DATA_BLOCK "DB_OrinCommandValidation"
{ S7_Optimized_Access := 'TRUE' }
VERSION : 0.1
NON_RETAIN
   VAR
      Data : "UDT_CommandValidationStatus";
   END_VAR

BEGIN
END_DATA_BLOCK
